GLOBALCONSTANTS PWM_Konstanten (* Global constants *)
  (* Standard: 61499-1; Description: Copyright (c) 2026 Meisterschulen am Ostbahnhof This program and the accompanying materials are made available under the terms of the Eclipse Public License 2.0 which is available at https://www.eclipse.org/legal/epl-2.0/ SPDX-License-Identifier: EPL-2.0 *)
  (* Version 1.0, 2026-09-27, Franz Höpfinger, Meisterschulen am Ostbahnhof, initial implementation - bisher an mehreren Stellen als Rohwert wiederholte PWM-Konstanten hierher ausgelagert: PWM_13BIT_SKALIERUNG (systemweit, keine Hardware-Korrektur) aus HebenSenken_ILOCK_QDA_PWM_OPC/Aufnahme_Automatik/Aufnahme_Entlastung_STG4; PWM_LASTTEILER_KORREKTUR (Korrekturfaktor speziell fuer die eingesetzte Danfoss-PVEA-Hardware) aus HebenSenken_ILOCK_QDA_PWM_OPC; VALUES_50_75_25_FACTOR_75/_25 (Multimeter-kalibrierte Korrekturfaktoren) neu aus values_50_75_25 v1.2 ausgelagert. *)
  PACKAGE MyLib::sys::const;
  VAR_GLOBAL CONSTANT
    PWM_13BIT_SKALIERUNG : REAL := REAL#81.91; (* Systemweit, KEIN Hardware-Korrekturfaktor: 0-100% -> 0-8191 (13-Bit-PWM-Register, PWM 13 Bit Normierung.pdf: Faktor = 8191/100) *)
    PWM_LASTTEILER_KORREKTUR : REAL := REAL#0.715; (* Korrekturfaktor speziell fuer die eingesetzte Danfoss-PVEA-Hardware (Lastteiler), Multimeter-kalibriert - siehe HebenSenken_ILOCK_QDA_PWM_OPC *)
    VALUES_50_75_25_FACTOR_75 : REAL := REAL#1.6; (* Multimeter-kalibrierter Korrekturfaktor auf die nominelle OUT_75-Spanne (25.0) in values_50_75_25 - Default ergibt den bisherigen eingebackenen Wert 40.0 (=25.0*1.6) *)
    VALUES_50_75_25_FACTOR_25 : REAL := REAL#1.4; (* Multimeter-kalibrierter Korrekturfaktor auf die nominelle OUT_25-Spanne (25.0) in values_50_75_25 - Default ergibt den bisherigen eingebackenen Wert 35.0 (=25.0*1.4) *)
  END_VAR
END_GLOBALCONSTANTS
